{attribute 'linkalways'} 
{attribute 'no_explicit_call' := 'This FB is a CLASS and must be accessed using methods or properties'}
{attribute 'enable_dynamic_creation'}
FUNCTION_BLOCK Node_F_VN_MaxElementElementwise_REAL EXTENDS VisionNode
VAR
    ipContainer : _ITcVnContainer;
    fMax : _REAL(0.0);
    hrPrev : _HRESULT(S_OK);
    hresult : _HRESULT(S_OK);
END_VAR

METHOD PUBLIC  Clone : I_Node
VAR
	pNode : POINTER TO Node_F_VN_MaxElementElementwise_REAL;
END_VAR
pNode := __NEW(Node_F_VN_MaxElementElementwise_REAL);
Clone := pNode^;
END_METHOD

METHOD FB_init : BOOL
VAR_INPUT
	bInitRetains : BOOL; // if TRUE, the retain variables are initialized (warm start / cold start)
	bInCopyCode : BOOL;  // if TRUE, the instance afterwards gets moved into the copy code (online change)
END_VAR
AddInput('ipContainer', ipContainer);
AddInput('hrPrev', hrPrev);
AddOutput('ipContainer', ipContainer);
AddOutput('fMax', fMax);
AddOutput('hresult',hresult);
END_METHOD

METHOD PROTECTED OnExecute
hresult.Value := F_VN_MaxElementElementwise_REAL(
    ipContainer := ipContainer.Value,
    fMax := fMax.Value,
    hrPrev:= hrPrev.Value);
END_METHOD

METHOD PUBLIC PreExecutionCheck
VAR_INPUT
	Check : I_PreExecutionChecks;
END_VAR
Check.IsTrue(ipContainer.IsValid, 'ipContainer must be a valid container');
Check.IsTrue(ipContainer.IsType(TC_GLOBAL_CONST_LIST.ContainerType_Vector_REAL), 'ipContainer contains incorrect type');
END_METHOD

END_FUNCTION_BLOCK

(* stored: Version 1.1.0.1, ProductVersion 3.1.4026.13
   POU Node_F_VN_MaxElementElementwise_REAL: Id {f915c4cc-9fb3-4daf-b229-5712475bdf98}, SpecialFunc None
   Folder Constructor: Id {c35299c1-465c-4e33-aa87-c6a6ae250af9}
   Method Clone: Id {d5ec640f-17b0-490b-9a7c-8ca47b2c4854}
   Method FB_init: Id {0a8fe3a7-a133-44f2-b79c-f95a7f211f25}
   Method OnExecute: Id {f54b3da6-dde2-474c-89ad-e9b3fc65bd7e}
   Method PreExecutionCheck: Id {a6ed43bc-ea86-4a24-a41b-775c2bac3235} *)
